// TwinCAT 3 PLC project AbstactDataStructures
// Title: Abstarct Data Structures
// Company: FisoThemes
// Author: Goodwill Mzumala
// Description: Exploring Abstract Data Structures in Structured Text for use in PLCs
// ProgramVersion: 3.1.4022.7
// libraries:
//   Tc2_Standard, * (Beckhoff Automation GmbH)
//   Tc2_System, * (Beckhoff Automation GmbH)
//   Tc2_Utilities, * (Beckhoff Automation GmbH)
//   Tc3_Module, * (Beckhoff Automation GmbH)
//   VisuSymbols,3.5.10.0,System
// project tree:
//   DUTs/Alias/ T_DATA_TYPE.TcDUT (not stored)
//   DUTs/Enum/ E_TYPE_CLASS.TcDUT
//   DUTs/Interface/ I_Stack.TcIO, I_Linked_List.TcIO, I_Queue.TcIO
//   DUTs/Struct/ ST_NODE.TcDUT
//   / GlobalTextList.TcGTLO, PlcTask.TcTTO (not stored)
//   POUs/Dynamic Array/Function Blocks/ FB_Dynamic_Array.TcPOU
//   POUs/Dynamic Array/Programs/ P_Dynamic_Array.TcPOU
//   POUs/Linked List/Function Blocks/ FB_Circular_Linked_List.TcPOU, FB_Doubly_Linked_List.TcPOU, FB_Singly_Linked_List.TcPOU
//   POUs/Linked List/Programs/ P_Doubly_Linked_List.TcPOU, P_Linked_List.TcPOU (not stored), P_Singly_Linked_List.TcPOU
//   POUs/ MAIN.TcPOU
//   POUs/Queue/Function Blocks/ FB_Dynamic_Array_Queue.TcPOU, FB_Linked_List_Queue.TcPOU
//   POUs/Queue/Programs/ P_Dynamic_Array_Queue.TcPOU, P_Linked_List_Queue.TcPOU, P_Queue.TcPOU
//   POUs/Stack/Function Blocks/ FB_Linked_List_Stack.TcPOU, FB_Dynamic_Array_Stack.TcPOU
//   POUs/Stack/Programs/ P_Dynamic_Array_Stack.TcPOU, P_Linked_List_Stack.TcPOU, P_Stack.TcPOU
// real-time tasks:
//   TASK PlcTask: cycle T#10ms, priority 20, ADS port 350

// ---- DUTs/Enum/E_TYPE_CLASS.TcDUT
// List of __SYSTEM.TYPE_CLASS.<type> used for reference
//{attribute 'qualified_only'}
{attribute 'strict'}
TYPE E_TYPE_CLASS :
(
	TYPE_BOOL 			:= DWORD#0,
    TYPE_BIT 			:= DWORD#1,
    TYPE_BYTE 			:= DWORD#2,
    TYPE_WORD 			:= DWORD#3,
    TYPE_DWORD 			:= DWORD#4,
    TYPE_LWORD 			:= DWORD#5,
    TYPE_SINT 			:= DWORD#6,
    TYPE_INT 			:= DWORD#7,
    TYPE_DINT 			:= DWORD#8,
    TYPE_LINT 			:= DWORD#9,
    TYPE_USINT 			:= DWORD#10,
    TYPE_UINT 			:= DWORD#11,
    TYPE_UDINT 			:= DWORD#12,
    TYPE_ULINT 			:= DWORD#13,
    TYPE_REAL 			:= DWORD#14,
    TYPE_LREAL 			:= DWORD#15,
    TYPE_STRING 		:= DWORD#16,
    TYPE_WSTRING 		:= DWORD#17,
    TYPE_TIME 			:= DWORD#18,
    TYPE_DATE 			:= DWORD#19,
    TYPE_DATEANDTIME 	:= DWORD#20,
    TYPE_TIMEOFDAY 		:= DWORD#21,
    TYPE_POINTER 		:= DWORD#22,
    TYPE_REFERENCE 		:= DWORD#23,
    TYPE_SUBRANGE 		:= DWORD#24,
    TYPE_ENUM 			:= DWORD#25,
    TYPE_ARRAY 			:= DWORD#26,
    TYPE_PARAMS 		:= DWORD#27,
    TYPE_USERDEF 		:= DWORD#28,
    TYPE_NONE 			:= DWORD#29,
    TYPE_ANY 			:= DWORD#30,
    TYPE_ANYBIT 		:= DWORD#31,
    TYPE_ANYDATE 		:= DWORD#32,
    TYPE_ANYINT 		:= DWORD#33,
    TYPE_ANYNUM 		:= DWORD#34,
    TYPE_ANYREAL 		:= DWORD#35,
    TYPE_LAZY 			:= DWORD#36,
    TYPE_LTIME 			:= DWORD#37,
    TYPE_BITCONST 		:= DWORD#38
)DWORD;
END_TYPE

// ---- DUTs/Struct/ST_NODE.TcDUT
{attribute 'enable_dynamic_creation'}
TYPE ST_NODE :
STRUCT
	pPrevious 	: POINTER TO ST_NODE := NULL; // Pointer to previos node.
	Data 		: T_DATA_TYPE;
	pNext 		: POINTER TO ST_NODE := NULL; // Pointer to next node.
END_STRUCT
END_TYPE

// ---- DUTs/Interface/I_Stack.TcIO
INTERFACE I_Stack

// Empties/Clears/Deletes all elements on the stack
METHOD Empty
END_METHOD

METHOD FB_exit : BOOL
VAR_INPUT
	bInCopyCode : BOOL; // if TRUE, the exit method is called for exiting an instance that is copied afterwards (online change).
END_VAR
END_METHOD

// Checks of stack is empty.
METHOD Is_Empty : BOOL
VAR_INPUT
END_VAR
END_METHOD

// Gets element at any position of the stack, wuthout removing it.
METHOD Peek : T_DATA_TYPE
VAR_INPUT
	nPosition : DINT;
END_VAR
END_METHOD

// Deletes/pops an element at the front of the stack 
METHOD Pop : T_DATA_TYPE
END_METHOD

// Adds/pushes an element to the front of the stack 
METHOD Push
VAR_INPUT
	Data 	: T_DATA_TYPE;
END_VAR
END_METHOD

// Traverse the stack and display each element as an array
METHOD Show
VAR_IN_OUT
	aList 		: ARRAY[*] OF T_DATA_TYPE; // Array to display data in list.
END_VAR
END_METHOD

// Gets size of the stack
METHOD Size : DINT;
END_METHOD

// Reads/returns the data at the top of the stack without removing it.
METHOD Top : T_DATA_TYPE
VAR_INPUT
END_VAR
END_METHOD

END_INTERFACE

// ---- DUTs/Interface/I_Linked_List.TcIO
INTERFACE I_Linked_List

// Creates/Adds an node to the end of the list
METHOD Create
VAR_INPUT
	Data : T_DATA_TYPE; // Data to add to new node.
END_VAR
END_METHOD

// Empties/Clears/Deletes list
METHOD Empty
END_METHOD

METHOD FB_exit : BOOL
VAR_INPUT
	bInCopyCode : BOOL; // if TRUE, the exit method is called for exiting an instance that is copied afterwards (online change).
END_VAR
END_METHOD

METHOD FB_init : BOOL
VAR_INPUT
	bInitRetains : BOOL; // if TRUE, the retain variables are initialized (warm start / cold start)
	bInCopyCode : BOOL;  // if TRUE, the instance afterwards gets moved into the copy code (online change)
END_VAR
END_METHOD

// Inserts node at a specific position in the list
METHOD Insert
VAR_INPUT
	Data 		: T_DATA_TYPE; 	// Data to add to new node.
	nPosition 	: DINT;		// Position to add new node in list.
END_VAR
END_METHOD

// Checks of list is empty.
METHOD Is_Empty : BOOL
VAR_INPUT
END_VAR
END_METHOD

// Gets element at any position of the list, wuthout removing it.
METHOD Peek : T_DATA_TYPE
VAR_INPUT
	nPosition : DINT;
END_VAR
END_METHOD

// Deletes/pops a node at the front of the list 
METHOD Pop : T_DATA_TYPE
END_METHOD

// Adds/pushes a node at the front of the list 
METHOD Push
VAR_INPUT
		Data 	: T_DATA_TYPE;
END_VAR
END_METHOD

// Deletes node at a specific position in the list
METHOD Remove : T_DATA_TYPE
VAR_INPUT
	nPosition 	: DINT; // Position of node to delete.
END_VAR
END_METHOD

// Reverse list
METHOD Reverse
END_METHOD

// Searches list for the first instance of data and returns it's location and whether it's in the list.
METHOD Search : BOOL
VAR_INPUT
	Data : T_DATA_TYPE; // Data to find in list
END_VAR
VAR_OUTPUT
	nPosition : DINT; // Location of the data  starting from 0. -1 means data is not found in list
END_VAR
END_METHOD

// Traverse the list to display each node
METHOD Show
VAR_IN_OUT
	aList 		: ARRAY[*] OF T_DATA_TYPE; // Array to display data in list.
END_VAR
END_METHOD

// Gets size of the list
METHOD Size : DINT;
END_METHOD

END_INTERFACE

// ---- DUTs/Interface/I_Queue.TcIO
INTERFACE I_Queue

(* Removes element from the front of the queue. *)
METHOD Dequeue : T_DATA_TYPE
VAR_INPUT
END_VAR
END_METHOD

(* Empties/Clears/Deletes all elements on the stack. *)
METHOD Empty
END_METHOD

(* Adds element to the rear of the queue. *)
METHOD Enqueue
VAR_INPUT
	Data 	: T_DATA_TYPE;
END_VAR
END_METHOD

METHOD FB_exit : BOOL
VAR_INPUT
	bInCopyCode : BOOL; // if TRUE, the exit method is called for exiting an instance that is copied afterwards (online change).
END_VAR
END_METHOD

METHOD FB_init : BOOL
VAR_INPUT
	bInitRetains : BOOL; // if TRUE, the retain variables are initialized (warm start / cold start)
	bInCopyCode : BOOL;  // if TRUE, the instance afterwards gets moved into the copy code (online change)
END_VAR
END_METHOD

(* Checks of queue is empty. *)
METHOD Is_Empty : BOOL
VAR_INPUT
END_VAR
END_METHOD

// Gets element at any position of the queue, without removing it.
METHOD Peek : T_DATA_TYPE
VAR_INPUT
	nPosition : DINT;
END_VAR
END_METHOD

(* Traverse the queue and display each element as an array. *)
METHOD Show
VAR_IN_OUT
	aList : ARRAY[*] OF T_DATA_TYPE; // Array to display data in list.
END_VAR
END_METHOD

(* Gets size of the queue. *)
METHOD Size : DINT;
END_METHOD

END_INTERFACE

// ---- POUs/Dynamic Array/Function Blocks/FB_Dynamic_Array.TcPOU
FUNCTION_BLOCK FB_Dynamic_Array
VAR_INPUT
	
END_VAR
VAR_OUTPUT
END_VAR
VAR
	pData 	: POINTER TO T_DATA_TYPE;
	nLength : DINT;
	t_Null	: T_DATA_TYPE;
END_VAR

(* Get element in array from specified poisiton. *)
METHOD Access : T_DATA_TYPE
VAR_INPUT
	nPosition : DINT;  // Position of element in dynamic array, 0 indexed.
END_VAR
IF nPosition < 0 THEN Access := t_Null; RETURN; END_IF
IF THIS^.Is_Empty() THEN FB_Init(FALSE,FALSE,(nPosition+1)*2); END_IF
IF nPosition >= THIS^.Size() THEN THIS^.Insert(t_Null, nPosition); END_IF
Access := THIS^.pData[nPosition];
END_METHOD

(* Deletes array from memory. *)
METHOD Clear
VAR_INPUT
END_VAR
IF NOT(THIS^.Is_Empty()) THEN __DELETE(THIS^.pData); THIS^.Is_Empty(); END_IF
END_METHOD

METHOD FB_exit : BOOL
VAR_INPUT
	bInCopyCode : BOOL; // if TRUE, the exit method is called for exiting an instance that is copied afterwards (online change).
END_VAR
THIS^.Clear();
END_METHOD

METHOD FB_init : BOOL
VAR_INPUT
	bInitRetains 	: BOOL; // if TRUE, the retain variables are initialized (warm start / cold start)
	bInCopyCode 	: BOOL;  // if TRUE, the instance afterwards gets moved into the copy code (online change)
	nLength 		: DINT; 	// Length to initialize array with, default is 10;
END_VAR
THIS^.Clear();
IF nLength > 0 THEN THIS^.pData := __NEW(T_DATA_TYPE, TO_UDINT(nLength)); END_IF
THIS^.nLength := nLength;
END_METHOD

(* Insert element into array at specified position. *)
METHOD Insert
VAR_INPUT
	Data 		: T_DATA_TYPE; 	// Data to insert in dynamic array.
	nPosition 	: DINT; 		// Position to insert data at in the dynamic array, 0 indexed. 
END_VAR
VAR
	pTemp_Data 		: POINTER TO T_DATA_TYPE;
	nTemp_Length 	: DINT;
	i 				: DINT;
END_VAR
IF nPosition < 0 THEN RETURN; END_IF
IF THIS^.Is_Empty() THEN FB_Init(FALSE,FALSE,(nPosition+1)*2); END_IF
IF nPosition < THIS^.Size() THEN 
	THIS^.pData[nPosition] := Data;
ELSE 
	THIS^.Resize((nPosition+1)*2);
	THIS^.pData[nPosition] := Data;
	END_IF
END_METHOD

(* Checks if array is empty. *)
METHOD Is_Empty : BOOL
VAR_INPUT
END_VAR
Is_Empty := THIS^.pData = 0;
IF Is_Empty THEN THIS^.nLength := 0; END_IF
END_METHOD

(* Manually resize dynamic array length. If Array become smaller, elements higher positions will be deleted. *)
METHOD Resize
VAR_INPUT
	nLength 		: DINT; // New length of dynamic array.
END_VAR
VAR_INST
	pTemp_Data 		: POINTER TO T_DATA_TYPE;
	nTemp_Length 	: DINT;
	i 				: DINT;
END_VAR
IF nLength <= 0 THEN THIS^.Clear(); RETURN; END_IF
IF THIS^.Is_Empty() THEN FB_init(FALSE,FALSE,nLength); RETURN; END_IF
IF THIS^.nLength = nLength THEN RETURN; END_IF

pTemp_Data 		:= THIS^.pData; 

nTemp_Length 	:= THIS^.nLength;
THIS^.nLength 	:= nLength;

THIS^.pData := __NEW(T_DATA_TYPE, TO_UDINT(THIS^.nLength));
FOR i := 0 TO TO_DINT(nTemp_Length-1) DO 
	IF i > TO_DINT(THIS^.nLength-1) THEN EXIT; END_IF 
	THIS^.pData[i] := pTemp_Data[i]; 
	END_FOR
__DELETE(pTemp_Data);
END_METHOD

(* Display elements in dynamic array in a static array. *)
METHOD Show
VAR_IN_OUT
	aList : ARRAY[*] OF T_DATA_TYPE; // Static array to display data in dynamic array.
END_VAR
VAR
	i,j : DINT;
END_VAR
FOR i := LOWER_BOUND(aList, 1) TO UPPER_BOUND(aList, 1) DO
	IF (j < TO_DINT(THIS^.Size())) AND NOT(THIS^.Is_Empty()) THEN
		aList[i] := THIS^.pData[j];
		j := j + 1; 
	ELSE 
		aList[i] := t_Null;
	 	END_IF
	END_FOR
END_METHOD

(* Gets the length of dynamic array. *)
METHOD Size : DINT
VAR_INPUT
END_VAR
Is_Empty(); Size := THIS^.nLength;
END_METHOD

END_FUNCTION_BLOCK

// ---- POUs/Dynamic Array/Programs/P_Dynamic_Array.TcPOU
PROGRAM P_Dynamic_Array
VAR
	bIs_Empty, bInsert, bAdd, bAccess, bResize, bClear : BOOL;
	nDyn_Size 	: DINT;
	aArray 		: ARRAY[0..30] OF T_DATA_TYPE;
	t_Access 	: T_DATA_TYPE;  
	fbDyn_Array : FB_Dynamic_Array(10);
	i 			: DINT;
END_VAR

bIs_Empty := fbDyn_Array.Is_Empty();
nDyn_Size := fbDyn_Array.Size();
fbDyn_Array.Show(aArray);

IF bInsert THEN
	fbDyn_Array.Insert(53476,0); 
	FOR i := 1 TO 9 DO fbDyn_Array.Insert(TO_ULINT(i*11),i); END_FOR
	bInsert := 0;
	END_IF
IF bAdd 	THEN fbDyn_Array.Insert(33,10); bAdd 	:= 0; END_IF
IF bAccess 	THEN t_Access := fbDyn_Array.Access(2); bAccess := 0; END_IF
IF bResize 	THEN fbDyn_Array.Resize(5); 			bResize := 0; END_IF
IF bClear 	THEN fbDyn_Array.Clear();				bClear 	:= 0; END_IF

END_PROGRAM

// ---- POUs/Linked List/Function Blocks/FB_Circular_Linked_List.TcPOU
FUNCTION_BLOCK FB_Circular_Linked_List IMPLEMENTS I_Linked_List
VAR_INPUT
END_VAR
VAR_OUTPUT
END_VAR
VAR
END_VAR

{warning 'add method implementation '}
(* Creates/Adds an node to the end of the list*)
METHOD Create
VAR_INPUT
	(* Data to add to new node.*)
	Data	: T_DATA_TYPE;
END_VAR
END_METHOD

{warning 'add method implementation '}
(* Empties/Clears/Deletes list*)
METHOD Empty
	pTemp	: POINTER TO ST_NODE;
END_METHOD

{warning 'add method implementation '}
(* Initializes or create an empty list*)
METHOD Init
END_METHOD

{warning 'add method implementation '}
(* Inserts node at a specific position in the list*)
METHOD Insert
VAR_INPUT
	(* Data to add to new node.*)
	Data	: T_DATA_TYPE;
	(* Position to add new node in list.*)
	nPosition	: UXINT;
END_VAR
END_METHOD

{warning 'add method implementation '}
METHOD Pop
END_METHOD

{warning 'add method implementation '}
METHOD Push
VAR_INPUT
	Data	: T_DATA_TYPE;
END_VAR
END_METHOD

{warning 'add method implementation '}
(* Deletes node at a specific position in the list*)
METHOD Remove
VAR_INPUT
	(* Position of node to delete.*)
	nPosition	: UXINT;
END_VAR
END_METHOD

{warning 'add method implementation '}
(* Searches list for the first instance of data and returns it's location and whether it's in the list.*)
METHOD Search : BOOL
VAR_INPUT
	(* Data to find in list*)
	Data	: T_DATA_TYPE;
END_VAR
VAR_OUTPUT
	(* Location of the data  starting from 1. 0 means data is not found in list*)
	nPosition	: UXINT;
END_VAR
END_METHOD

{warning 'add method implementation '}
METHOD Show
END_METHOD

{warning 'add method implementation '}
(* Gets size of the list*)
METHOD Size : UXINT
END_METHOD

END_FUNCTION_BLOCK

// ---- POUs/Linked List/Function Blocks/FB_Doubly_Linked_List.TcPOU
FUNCTION_BLOCK FB_Doubly_Linked_List IMPLEMENTS I_Linked_List
VAR
	pHead :  POINTER TO ST_NODE;
	pTail :  POINTER TO ST_NODE;
	t_Null: T_DATA_TYPE;
END_VAR

(* Creates/Adds an node to the end of the list. *)
METHOD Create
VAR_INPUT
	(* Data to add to new node.*)
	Data		: T_DATA_TYPE;
END_VAR
VAR
	pTemp 		:  POINTER TO ST_NODE; //  New node will be allocated at this pointer
	pPrevious 	: POINTER TO ST_NODE; // Previous node location will be stored at this pointer temporarily
END_VAR
pTemp := __NEW(ST_NODE);
pTemp^.Data := Data;
IF THIS^.pHead = 0 THEN 
	THIS^.pHead := pTemp; 
	THIS^.pTail := THIS^.pHead; // If the pointer to the pHead is NULL then give it an address. The pTail address of the first node is the pHead.
ELSE
	pPrevious := THIS^.pTail;
	THIS^.pTail^.pNext := pTemp; 
	THIS^.pTail := pTemp;
	THIS^.pTail^.pPrevious := pPrevious; 
	END_IF // Point previous node's pNext to the address of pTemp and set pTail to pTemp.
END_METHOD

(* Empties/Clears/Deletes list*)
METHOD Empty
VAR
	pTemp : POINTER TO ST_NODE;
END_VAR
pTail := 0;
pTemp := pHead;
WHILE pTemp <> 0 DO
	pTemp := pTemp^.pNext; THIS^.Pop();
END_WHILE
END_METHOD

METHOD FB_exit : BOOL
VAR_INPUT
	(* if TRUE, the exit method is called for exiting an instance that is copied afterwards (online change).*)
	bInCopyCode	: BOOL;
END_VAR
This^.Empty();
END_METHOD

METHOD FB_init : BOOL
VAR_INPUT
	(* if TRUE, the retain variables are initialized (warm start / cold start)*)
	bInitRetains	: BOOL;
	(* if TRUE, the instance afterwards gets moved into the copy code (online change)*)
	bInCopyCode	: BOOL;
END_VAR
END_METHOD

(* Inserts node at a specific position in the list*)
METHOD Insert
VAR_INPUT
	(* Data to add to new node.*)
	Data	: T_DATA_TYPE;
	(* Position to add new node in list.*)
	nPosition	: DINT;
END_VAR
END_METHOD

(* Checks of list is empty.*)
METHOD Is_Empty : BOOL
END_METHOD

(* Gets element at any position of the list, wuthout removing it.*)
METHOD Peek : T_DATA_TYPE
VAR_INPUT
	nPosition	: DINT;
END_VAR
END_METHOD

(* Deletes/pops a node at the front of the list *)
METHOD Pop : T_DATA_TYPE
VAR
	pTemp : POINTER TO ST_NODE;
END_VAR
IF THIS^.pHead = 0 THEN RETURN; END_IF 
Pop := pHead^.Data;
pTemp := pHead^.pNext;
__DELETE(pHead);
pHead := pTemp;
END_METHOD

(* Adds/pushes a node at the front of the list *)
METHOD Push
VAR_INPUT
	Data	: T_DATA_TYPE;
END_VAR
END_METHOD

(* Deletes node at a specific position in the list*)
METHOD Remove : T_DATA_TYPE
VAR_INPUT
	(* Position of node to delete.*)
	nPosition	: DINT;
END_VAR
END_METHOD

(* Reverse list*)
METHOD Reverse
END_METHOD

//{warning 'add method implementation '}
(* Searches list for the first instance of data and returns it's location and whether it's in the list.*)
METHOD Search : BOOL
VAR_INPUT
	(* Data to find in list*)
	Data	: T_DATA_TYPE;
END_VAR
VAR_OUTPUT
	(* Location of the data  starting from 1. 0 means data is not found in list*)
	nPosition	: DINT;
END_VAR
END_METHOD

(* Traverse the list to display each node. *)
METHOD Show
VAR_IN_OUT
	aList 		: ARRAY[*] OF T_DATA_TYPE; // Array to display data in list.
END_VAR
VAR
	pCurrent 	: POINTER TO ST_NODE;
	i 			: DINT;
END_VAR
END_METHOD

(* Gets size of the list*)
METHOD Size : DINT
END_METHOD

END_FUNCTION_BLOCK

// ---- POUs/Linked List/Function Blocks/FB_Singly_Linked_List.TcPOU
// Linear/Singly Linked List
FUNCTION_BLOCK FB_Singly_Linked_List IMPLEMENTS I_Linked_List
VAR_INPUT
END_VAR
VAR_OUTPUT
END_VAR
VAR
	pHead :  POINTER TO ST_NODE;
	pTail :  POINTER TO ST_NODE;
	t_Null: T_DATA_TYPE;
END_VAR

// Creates/Adds an node to the end of the list
METHOD Create
VAR_INPUT
	Data : T_DATA_TYPE; // Data to add to new node.
END_VAR
VAR
	pTemp :  POINTER TO ST_NODE;
END_VAR
pTemp := __NEW(ST_NODE); 	// Allocate space in memory for a node.
pTemp^.Data := Data;		// Assign Data to the new node.
IF pHead = 0 THEN pHead := pTemp; pTail := pHead; // If the pointer to the pHead is NULL then give it an address. The pTail address of the first node is the pHead.
ELSE  pTail^.pNext := pTemp; pTail := pTail^.pNext; END_IF // Point previous node's pNext to the address of pTemp and set pTail to pTemp.
END_METHOD

// Empties/Clears/Deletes list
METHOD Empty
VAR
	pTemp : POINTER TO ST_NODE;
END_VAR
pTail := 0;
pTemp := pHead;
WHILE pTemp <> 0 DO
	pTemp := pTemp^.pNext; THIS^.Pop();
END_WHILE
END_METHOD

METHOD FB_exit : BOOL
VAR_INPUT
	bInCopyCode : BOOL; // if TRUE, the exit method is called for exiting an instance that is copied afterwards (online change).
END_VAR
Empty();
END_METHOD

// Initializes or create an empty list
METHOD Init
THIS^.Empty();
pHead := 0;
pTail := 0;
END_METHOD

// Inserts node at a specific position in the list
METHOD Insert
VAR_INPUT
	Data 		: T_DATA_TYPE; 	// Data to add to new node.
	nPosition 	: DINT;		// Position to add new node in list.
END_VAR
VAR
	pPrevious 	: POINTER TO ST_NODE;
	pCurrent 	: POINTER TO ST_NODE;
	pTemp 		: POINTER TO ST_NODE;
	i 			: DINT;
END_VAR
IF nPosition < 0 THEN RETURN; END_IF
IF nPosition = 0 THEN THIS^.Push(Data); RETURN; END_IF
pTemp := __NEW(ST_NODE);
pCurrent := THIS^.pHead;
FOR i := 1 TO nPosition DO // traverse
	pPrevious := pCurrent; 
	pCurrent := pPrevious^.pNext;
	IF pCurrent = 0 THEN EXIT; END_IF
	END_FOR;
pTemp^.Data := Data;
IF pPrevious <> 0 THEN pPrevious^.pNext := pTemp; END_IF
pTemp^.pNext := pCurrent;
END_METHOD

(* Checks of list is empty.*)
METHOD Is_Empty : BOOL
Is_Empty := pHead = 0;
END_METHOD

// Gets element at any position of the list. Returns 0 if element is not found
METHOD Peek : T_DATA_TYPE
VAR_INPUT
	nPosition : DINT;
END_VAR
VAR 
	i 		: DINT;
	pTemp 	: POINTER TO ST_NODE;
END_VAR
IF nPosition >= 0 AND nPosition < THIS^.Size() THEN
	pTemp := pHead;
	FOR i := 0 TO nPosition DO
		Peek := pTemp^.Data;
		pTemp := pTemp^.pNext;
		END_FOR
ELSE
	Peek := 0;
	END_IF
END_METHOD

// Deletes/pops a node at the start of the list 
METHOD Pop : T_DATA_TYPE
VAR
	pTemp : POINTER TO ST_NODE;
END_VAR
IF THIS^.pHead = 0 THEN RETURN; END_IF 
Pop := pHead^.Data;
pTemp := pHead^.pNext;
__DELETE(pHead);
pHead := pTemp;
END_METHOD

// Adds/pushes a node at the start of the list 
METHOD Push
VAR_INPUT
	Data 	: T_DATA_TYPE;
END_VAR
VAR
	pTemp 	:  POINTER TO ST_NODE;
END_VAR
pTemp := __NEW(ST_NODE);
pTemp^.Data := Data;
IF THIS^.pHead = 0 THEN THIS^.pHead := pTemp; THIS^.pTail := THIS^.pHead;
ELSE pTemp^.pNext := THIS^.pHead; THIS^.pHead := pTemp; END_IF
END_METHOD

// Deletes node at a specific position in the list
METHOD Remove : T_DATA_TYPE
VAR_INPUT
	nPosition 	: DINT; // Position of node to delete.
END_VAR
VAR
	pPrevious 	: POINTER TO ST_NODE;
	pCurrent 	: POINTER TO ST_NODE;
	i 			: DINT;
END_VAR
IF nPosition < 0 THEN RETURN; END_IF
pCurrent := pHead;
FOR i := 1 TO nPosition DO
	pPrevious := pCurrent;
	pCurrent := pCurrent^.pNext;
	END_FOR;
Remove := pCurrent^.Data;
pPrevious^.pNext := pCurrent^.pNext;
__DELETE(pCurrent);
END_METHOD

// Reverses list
METHOD Reverse
VAR
	pPrevious 	: POINTER TO ST_NODE;
	pCurrent 	: POINTER TO ST_NODE;
	pNext	 	: POINTER TO ST_NODE;
	i 			: DINT;
END_VAR
pCurrent := pHead;
pNext := pCurrent;
WHILE pCurrent <> 0 DO
	pNext := pNext^.pNext;
	pCurrent^.pNext := pPrevious;
	pPrevious := pCurrent;
	pCurrent := pNext;
END_WHILE
pHead := pPrevious;
END_METHOD

// Searches list for the first instance of data and returns it's location and whether it's in the list.
METHOD Search : BOOL
VAR_INPUT
	Data : T_DATA_TYPE; // Data to find in list
END_VAR
VAR_OUTPUT
	nPosition : DINT; // Location of the data  starting from 1. 0 means data is not found in list
END_VAR
VAR
	pTemp 	: POINTER TO ST_NODE;
	i 		: DINT;
END_VAR
pTemp := pHead;
WHILE pTemp <> 0 DO
	
	Search := pTemp^.Data = Data;
	IF Search THEN nPosition := i; EXIT; ELSE nPosition := 0; END_IF
	i := i + 1;
	pTemp := pTemp^.pNext;
END_WHILE
END_METHOD

// Traverse the list to display each node
METHOD Show
VAR_IN_OUT
	aList 		: ARRAY[*] OF T_DATA_TYPE; // Array to display data in list.
END_VAR
VAR
	pCurrent 	: POINTER TO ST_NODE;
	i 			: DINT;
END_VAR
pCurrent := THIS^.pHead;
FOR i := LOWER_BOUND(aList, 1) TO UPPER_BOUND(aList, 1) DO
	IF pCurrent <> 0 THEN 
		aList[i] := pCurrent^.Data; 
		pCurrent := pCurrent^.pNext;
	ELSE
		aList[i] := t_Null;
		END_IF
	END_FOR
END_METHOD

// Gets size of the list
METHOD Size : DINT;
VAR
	pTemp 	: POINTER TO ST_NODE;
	i 		: dINT;
END_VAR
pTemp := pHead;
WHILE pTemp <> 0 DO
	pTemp := pTemp^.pNext; i := i + 1;;
END_WHILE
Size := i;
END_METHOD

END_FUNCTION_BLOCK

// ---- POUs/Linked List/Programs/P_Doubly_Linked_List.TcPOU
PROGRAM P_Doubly_Linked_List
VAR
	nState 			: BYTE;
	fbLinked_List 	: FB_Doubly_Linked_List;
	Peek 			: T_DATA_TYPE;
	
	bFound 			: BOOL;		// Is data in the created list?
	nPosition 		: DINT;	// At what position is the data on the list? 0 means no data found. Head mode is 1.
	
	nSize 			: DINT; 	// Dispays size of list after it's created
	nDelete_Size 	: DINT; 	// Displays size of list after deleting an element.
	nInsert_Size 	: DINT; 	// Displays size of list after inserting an element.
	
	aArray 			: ARRAY[1..6] OF T_DATA_TYPE; // Displays created list.
	aDelete_Array 	: ARRAY[1..6] OF T_DATA_TYPE; // Displays list after deleting element at a position.
	aInsert_Array	: ARRAY[1..6] OF T_DATA_TYPE; // Displays list after inserting element at a position.
END_VAR

CASE nState OF 
	0: // Create list, display list, get list size and find an item in the list.
		fbLinked_List.Create(1);
		fbLinked_List.Create(2);
		fbLinked_List.Create(3);
		fbLinked_List.Create(4);
		fbLinked_List.Create(5);
		fbLinked_List.Show(aArray);
		Peek := fbLinked_List.Peek(1);
		nSize := fbLinked_List.Size();
		bFound := fbLinked_List.Search(Data := 5, nPosition => nPosition);

		nState := nState + 1;			
	
	1: // Remove an elements from the list, display list and get the list size
		fbLinked_list.Remove(3);
		fbLinked_List.Pop();
		fbLinked_List.Show(aDelete_Array);
		nDelete_Size := fbLinked_List.Size();
	
		nState := nState + 1;
	
	2: // Insert elements into list, display it and the list size
		fbLinked_List.Push(11);
		fbLinked_List.Insert(14,3);
		fbLinked_List.Show(aInsert_Array);
		nInsert_Size := fbLinked_List.Size();
		
		nState := nState + 1;
		
	3: // Clear list, then finish.
		fbLinked_List.Empty();
		
		nState := nState + 1;
END_CASE

END_PROGRAM

// ---- POUs/Linked List/Programs/P_Singly_Linked_List.TcPOU
PROGRAM P_Singly_Linked_List
VAR
	nState 			: BYTE;
	fbLinked_List 	: FB_Singly_Linked_List;
	Peek 			: T_DATA_TYPE;
	
	bFound 			: BOOL;		// Is data in the created list?
	nPosition 		: DINT;	// At what position is the data on the list? 0 means no data found. Head mode is 1.
	
	nCreate_Size 	: DINT; 	// Dispays size of list after it's created
	nDelete_Size 	: DINT; 	// Displays size of list after deleting an element.
	nInsert_Size 	: DINT; 	// Displays size of list after inserting an element.
	nClear_Size 	: DINT; 	// Displays size of list after clearing all elements.
	
	aCreate_Array 	: ARRAY[1..6] OF T_DATA_TYPE; // Displays created list.
	aDelete_Array 	: ARRAY[1..6] OF T_DATA_TYPE; // Displays list after deleting element at a position.
	aInsert_Array	: ARRAY[1..6] OF T_DATA_TYPE; // Displays list after inserting element at a position.
	aClear_Array	: ARRAY[1..6] OF T_DATA_TYPE; // Displays list after clearing all elements.
	
	
END_VAR

CASE nState OF 
	0: // Create list, display list, get list size and find an item in the list.
		fbLinked_List.Create(1);
		fbLinked_List.Create(2);
		fbLinked_List.Create(3);
		fbLinked_List.Create(4);
		fbLinked_List.Create(5);
		fbLinked_List.Show(aCreate_Array);
		Peek := fbLinked_List.Peek(1);
		nCreate_Size := fbLinked_List.Size();
		bFound := fbLinked_List.Search(Data := 5, nPosition => nPosition);

		nState := nState + 1;			
	
	1: // Remove an elements from the list, display list and get the list size
		fbLinked_list.Remove(3);
		fbLinked_List.Pop();
		fbLinked_List.Show(aDelete_Array);
		nDelete_Size := fbLinked_List.Size();
	
		nState := nState + 1;
	
	2: // Insert elements into list, display it and the list size
		fbLinked_List.Push(11);
		fbLinked_List.Insert(14,3);
		fbLinked_List.Show(aInsert_Array);
		nInsert_Size := fbLinked_List.Size();
		
		nState := nState + 1;
		
	3: // Clear list, then finish.
		fbLinked_List.Empty();
		fbLinked_List.Show(aClear_Array);
		nClear_Size := fbLinked_List.Size();
		
		nState := nState + 1;
END_CASE

END_PROGRAM

// ---- POUs/MAIN.TcPOU
PROGRAM MAIN
VAR
END_VAR

P_Dynamic_Array();
P_Linked_List();
P_Queue();
P_Stack();

END_PROGRAM

// ---- POUs/Queue/Programs/P_Queue.TcPOU
PROGRAM P_Queue
VAR
END_VAR

P_Dynamic_Array_Queue();
P_Linked_List_Queue();

END_PROGRAM

// ---- POUs/Queue/Programs/P_Dynamic_Array_Queue.TcPOU
PROGRAM P_Dynamic_Array_Queue
VAR
	nState 	: BYTE;
	fbQueue : FB_Dynamic_Array_Queue;
	
	bInit_Is_Empty 		: BOOL;
	nInit_Size 			: DINT;
	Init_Peek 			: T_DATA_TYPE;
	aInit_Show 			: ARRAY[1..6] OF T_DATA_TYPE;
	
	bEnqueue_Is_Empty 	: BOOL;
	nEnqueue_Size 		: DINT;
	Enqueue_Peek 		: T_DATA_TYPE;
	aEnqueue_Show 		: ARRAY[1..6] OF T_DATA_TYPE;
	
	bDequeue_Is_Empty 	: BOOL;
	nDequeue_Size 		: DINT;
	Dequeue_Peek 		: T_DATA_TYPE;
	aDequeue_Show 		: ARRAY[1..6] OF T_DATA_TYPE;
	
	bEmpty_Is_Empty 	: BOOL;
	nEmpty_Size 		: DINT;
	Empty_Peek 			: T_DATA_TYPE;
	aEmpty_Show 		: ARRAY[1..6] OF T_DATA_TYPE;
END_VAR

CASE nState OF
	0: // Init
		bInit_Is_Empty := fbQueue.Is_Empty();
		nInit_Size :=  fbQueue.Size();
		Init_Peek := fbQueue.Peek(0);
		fbQueue.Show(aInit_Show);
		
		nState := nState + 1;
		
	1: // Enqueue elements
		fbQueue.Enqueue(1);
		fbQueue.Enqueue(2);
		fbQueue.Enqueue(3);
		fbQueue.Enqueue(4);
		fbQueue.Enqueue(5);
		bEnqueue_Is_Empty := fbQueue.Is_Empty();
		nEnqueue_Size := fbQueue.Size();
		Enqueue_Peek := fbQueue.Peek(0);
		fbQueue.Show(aEnqueue_Show);
		
		nState := nState + 1;
	
	2: // Dequeue elements
		fbQueue.Dequeue();
		fbQueue.Dequeue(); 
		bDequeue_Is_Empty := fbQueue.Is_Empty();
		nDequeue_Size := fbQueue.Size();
		Dequeue_Peek := fbQueue.Peek(0);
		fbQueue.Show(aDequeue_Show);
		
		nState := nState + 1;
	
	3: // Empty Queue
		fbQueue.Empty();
		bEmpty_Is_Empty := fbQueue.Is_Empty();
		nEmpty_Size := fbQueue.Size();
		Empty_Peek := fbQueue.Peek(0);
		fbQueue.Show(aEmpty_Show);
		
		nState := nState + 1;
	
END_CASE

END_PROGRAM

// ---- POUs/Queue/Function Blocks/FB_Dynamic_Array_Queue.TcPOU
FUNCTION_BLOCK FB_Dynamic_Array_Queue IMPLEMENTS I_Queue
VAR
	fbDynamic_Array : FB_Dynamic_Array(10);
	nSize 			: DINT;
END_VAR

(* Removes element from the front of the queue. *)
METHOD Dequeue : T_DATA_TYPE
VAR 
	i : DINT;
END_VAR
Dequeue := THIS^.fbDynamic_Array.Access(0);
IF THIS^.Is_Empty() THEN RETURN; END_IF
nSize := THIS^.Size() - 1;
FOR i := 1 TO THIS^.nSize DO
	THIS^.fbDynamic_Array.Insert(THIS^.fbDynamic_Array.Access(i),i-1);
	END_FOR
END_METHOD

(* Empties/Clears/Deletes all elements on the stack. *)
METHOD Empty
THIS^.fbDynamic_Array.Clear(); 
THIS^.nSize := THIS^.fbDynamic_Array.Size();
END_METHOD

(* Adds element to the rear of the queue. *)
METHOD Enqueue
VAR_INPUT
	Data	: T_DATA_TYPE;
END_VAR
nSize := THIS^.Size() + 1;
THIS^.fbDynamic_Array.Insert(Data, THIS^.Size()-1);
END_METHOD

METHOD FB_exit : BOOL
VAR_INPUT
	(* if TRUE, the exit method is called for exiting an instance that is copied afterwards (online change).*)
	bInCopyCode	: BOOL;
END_VAR
THIS^.Empty();
END_METHOD

METHOD FB_init : BOOL
VAR_INPUT
	(* if TRUE, the retain variables are initialized (warm start / cold start)*)
	bInitRetains	: BOOL;
	(* if TRUE, the instance afterwards gets moved into the copy code (online change)*)
	bInCopyCode	: BOOL;
END_VAR
END_METHOD

(* Checks of queue is empty. *)
METHOD Is_Empty : BOOL
Is_Empty := nSize = 0;
IF Is_Empty THEN THIS^.Empty(); END_IF
END_METHOD

(* Gets element at any position of the queue, without removing it.*)
METHOD Peek : T_DATA_TYPE
VAR_INPUT
	nPosition	: DINT;
END_VAR
IF (nPosition > THIS^.nSize - 1) THEN nPosition := -1; END_IF
Peek := THIS^.fbDynamic_Array.Access(nPosition);
END_METHOD

(* Traverse the queue and display each element as an array. *)
METHOD Show
VAR_IN_OUT
	aList : ARRAY[*] OF T_DATA_TYPE; // Array to display data in list.
END_VAR
VAR
	i,j : DINT;
END_VAR
FOR i := LOWER_BOUND(aList, 1) TO UPPER_BOUND(aList, 1) DO
	IF j < TO_DINT(THIS^.Size()) AND NOT(THIS^.Is_Empty())THEN 
		aList[i] := THIS^.fbDynamic_Array.Access(j);
		j := j + 1;
	ELSE 
		aList[i] := THIS^.fbDynamic_Array.Access(-1);
		END_IF
	END_FOR
END_METHOD

(* Gets size of the queue. *)
METHOD Size : DINT
IF NOT(THIS^.Is_Empty())THEN Size := THIS^.nSize; END_IF
END_METHOD

END_FUNCTION_BLOCK

// ---- POUs/Queue/Programs/P_Linked_List_Queue.TcPOU
PROGRAM P_Linked_List_Queue
VAR
	nState 	: BYTE;
	fbQueue : FB_Linked_List_Queue;
	
	bInit_Is_Empty 		: BOOL;
	nInit_Size 			: DINT;
	Init_Peek 			: T_DATA_TYPE;
	aInit_Show 			: ARRAY[1..6] OF T_DATA_TYPE;
	
	bEnqueue_Is_Empty 	: BOOL;
	nEnqueue_Size 		: DINT;
	Enqueue_Peek 		: T_DATA_TYPE;
	aEnqueue_Show 		: ARRAY[1..6] OF T_DATA_TYPE;
	
	bDequeue_Is_Empty 	: BOOL;
	nDequeue_Size 		: DINT;
	Dequeue_Peek 		: T_DATA_TYPE;
	aDequeue_Show 		: ARRAY[1..6] OF T_DATA_TYPE;
	
	bEmpty_Is_Empty 	: BOOL;
	nEmpty_Size 		: DINT;
	Empty_Peek 			: T_DATA_TYPE;
	aEmpty_Show 		: ARRAY[1..6] OF T_DATA_TYPE;
END_VAR

CASE nState OF
	0: // Init
		bInit_Is_Empty := fbQueue.Is_Empty();
		nInit_Size :=  fbQueue.Size();
		Init_Peek := fbQueue.Peek(0);
		fbQueue.Show(aInit_Show);
		
		nState := nState + 1;
		
	1: // Enqueue elements
		fbQueue.Enqueue(1);
		fbQueue.Enqueue(2);
		fbQueue.Enqueue(3);
		fbQueue.Enqueue(4);
		fbQueue.Enqueue(5);
		bEnqueue_Is_Empty := fbQueue.Is_Empty();
		nEnqueue_Size := fbQueue.Size();
		Enqueue_Peek := fbQueue.Peek(0);
		fbQueue.Show(aEnqueue_Show);
		
		nState := nState + 1;
	
	2: // Dequeue elements
		fbQueue.Dequeue();
		fbQueue.Dequeue(); 
		bDequeue_Is_Empty := fbQueue.Is_Empty();
		nDequeue_Size := fbQueue.Size();
		Dequeue_Peek := fbQueue.Peek(0);
		fbQueue.Show(aDequeue_Show);
		
		nState := nState + 1;
	
	3: // Empty Queue
		fbQueue.Empty();
		bEmpty_Is_Empty := fbQueue.Is_Empty();
		nEmpty_Size := fbQueue.Size();
		Empty_Peek := fbQueue.Peek(0);
		fbQueue.Show(aEmpty_Show);
		
		nState := nState + 1;
	
END_CASE

END_PROGRAM

// ---- POUs/Queue/Function Blocks/FB_Linked_List_Queue.TcPOU
FUNCTION_BLOCK FB_Linked_List_Queue IMPLEMENTS I_Queue
VAR
	fbLinked_List : FB_Singly_Linked_List;
END_VAR

(* Removes element from the front of the queue. *)
METHOD Dequeue : T_DATA_TYPE
Dequeue := THIS^.fbLinked_List.Pop();
END_METHOD

(* Empties/Clears/Deletes all elements on the stack. *)
METHOD Empty
THIS^.fbLinked_List.Empty();
END_METHOD

(* Adds element to the rear of the queue. *)
METHOD Enqueue
VAR_INPUT
	Data	: T_DATA_TYPE;
END_VAR
THIS^.fbLinked_List.Create(Data);
END_METHOD

METHOD FB_exit : BOOL
VAR_INPUT
	(* if TRUE, the exit method is called for exiting an instance that is copied afterwards (online change).*)
	bInCopyCode	: BOOL;
END_VAR
THIS^.Empty();
END_METHOD

METHOD FB_init : BOOL
VAR_INPUT
	(* if TRUE, the retain variables are initialized (warm start / cold start)*)
	bInitRetains	: BOOL;
	(* if TRUE, the instance afterwards gets moved into the copy code (online change)*)
	bInCopyCode	: BOOL;
END_VAR
END_METHOD

(* Checks of queue is empty. *)
METHOD Is_Empty : BOOL
Is_Empty := THIS^.fbLinked_List.Is_Empty();
END_METHOD

(* Gets element at any position of the queue, without removing it.*)
METHOD Peek : T_DATA_TYPE
VAR_INPUT
	nPosition	: DINT;
END_VAR
Peek := THIS^.fbLinked_List.Peek(nPosition);
END_METHOD

(* Traverse the queue and display each element as an array. *)
METHOD Show
VAR_IN_OUT
	aList :  ARRAY[*] OF T_DATA_TYPE; // Array to display data in list.
END_VAR
THIS^.fbLinked_List.Show(aList);
END_METHOD

(* Gets size of the queue. *)
METHOD Size : DINT
Size := THIS^.fbLinked_List.Size();
END_METHOD

END_FUNCTION_BLOCK

// ---- POUs/Stack/Programs/P_Stack.TcPOU
PROGRAM P_Stack
VAR
END_VAR

P_Dynamic_Array_Stack();
P_Linked_List_Stack();

END_PROGRAM

// ---- POUs/Stack/Programs/P_Dynamic_Array_Stack.TcPOU
PROGRAM P_Dynamic_Array_Stack
VAR
	nState 	: BYTE;
	fbStack : FB_Dynamic_Array_Stack;
	
	
	// Init
	bInit_Is_Empty 	: BOOL;
	nInit_Size 		: DINT;
	Init_Top 		: T_DATA_TYPE;
	aInit_Stack 	: ARRAY[1..6] OF T_DATA_TYPE;
	
	// Pust element to stack
	bPush_Is_Empty 	: BOOL;
	nPush_Size 		: DINT;
	Push_Top 		: T_DATA_TYPE;
	Push_Peek		: T_DATA_TYPE;
	aPush_Stack 	: ARRAY[1..6] OF T_DATA_TYPE; 
	
	// Pop element from stack
	bPop_Is_Empty 	: BOOL;
	nPop_Size 		: DINT;
	Pop_Top 		: T_DATA_TYPE;
	aPop_Stack 		: ARRAY[1..6] OF T_DATA_TYPE; 
	
	// Empty Stack
	bEmpty_Is_Empty : BOOL;
	nEmpty_Size 	: DINT;
	Empty_Top 		: T_DATA_TYPE;
	aEmpty_Stack 	: ARRAY[1..6] OF T_DATA_TYPE; 
END_VAR

CASE nState OF
	0: // Init
		bInit_Is_Empty := fbStack.Is_Empty();
		nInit_Size :=  fbStack.Size();
		Init_Top := fbStack.Top();
		fbStack.Show(aInit_Stack);
		
		nState := nState + 1;
		
	1: // Push Element to tack
		fbStack.Push(1);
		fbStack.Push(2);
		fbStack.Push(3);
		fbStack.Push(4);
		fbStack.Push(5);
		bPush_Is_Empty := fbStack.Is_Empty();
		nPush_Size := fbStack.Size();
		Push_Top := fbStack.Top();
		Push_Peek := fbStack.Peek(2);
		fbStack.Show(aPush_Stack);
		
		nState := nState + 1;
	
	2: // Pop elements from stack
		fbStack.Pop();
		fbStack.Pop();
		bPop_Is_Empty := fbStack.Is_Empty();
		nPop_Size := fbStack.Size();
		Pop_Top := fbStack.Top();
		fbStack.Show(aPop_Stack);
		
		nState := nState + 1;
		
	3: // Empty stack
		fbStack.Empty();
		bEmpty_Is_Empty := fbStack.Is_Empty();
		nEmpty_Size := fbStack.Size();
		Empty_Top := fbStack.Top();
		fbStack.Show(aEmpty_Stack);
		
		nState := nState + 1;
END_CASE

END_PROGRAM

// ---- POUs/Stack/Function Blocks/FB_Dynamic_Array_Stack.TcPOU
FUNCTION_BLOCK FB_Dynamic_Array_Stack IMPLEMENTS I_Stack
VAR_INPUT
END_VAR
VAR_OUTPUT
END_VAR
VAR
	fbDynamic_Array : FB_Dynamic_Array(10); 
	nTop_Index 		: DINT; 
	nSize 			: DINT;
	t_Null 			: T_DATA_TYPE;
END_VAR

(* Empties/Clears/Deletes all elements on the stack*)
METHOD Empty
THIS^.fbDynamic_Array.Clear(); 
THIS^.nSize := THIS^.fbDynamic_Array.Size();
END_METHOD

METHOD FB_exit : BOOL
VAR_INPUT
	(* if TRUE, the exit method is called for exiting an instance that is copied afterwards (online change).*)
	bInCopyCode	: BOOL;
END_VAR
THIS^.Empty();
END_METHOD

METHOD FB_init : BOOL
VAR_INPUT
	bInitRetains : BOOL; // if TRUE, the retain variables are initialized (warm start / cold start)
	bInCopyCode : BOOL;  // if TRUE, the instance afterwards gets moved into the copy code (online change)
END_VAR
END_METHOD

(* Checks of stack is empty.*)
METHOD Is_Empty : BOOL
Is_Empty := nSize = 0;
IF Is_Empty THEN THIS^.Empty(); END_IF
END_METHOD

(* Gets element at any position of the stack, without removing it.*)
METHOD Peek : T_DATA_TYPE
VAR_INPUT
	nPosition	: DINT;
END_VAR
IF (nPosition > THIS^.nSize - 1) THEN nPosition := -1; END_IF
Peek := THIS^.fbDynamic_Array.Access(nPosition);
END_METHOD

(* Deletes/pops an element at the front of the stack *)
METHOD Pop : T_DATA_TYPE
Pop := THIS^.fbDynamic_Array.Access(THIS^.Size() - 1);
IF NOT(THIS^.Is_Empty()) THEN nSize := THIS^.Size() - 1; END_IF
END_METHOD

(* Adds/pushes an element to the front of the stack *)
METHOD Push
VAR_INPUT
	Data	: T_DATA_TYPE;
END_VAR
nSize := THIS^.Size() + 1;
THIS^.fbDynamic_Array.Insert(Data, THIS^.Size()-1);
END_METHOD

(* Traverse the stack and display each element as an array. *)
METHOD Show
VAR_IN_OUT
	aList : ARRAY[*] OF T_DATA_TYPE; // Array to display data in list.
END_VAR
VAR
	i,j : DINT;
END_VAR
FOR i := LOWER_BOUND(aList, 1) TO UPPER_BOUND(aList, 1) DO
	IF j < TO_DINT(THIS^.Size()) AND NOT(THIS^.Is_Empty())THEN 
		aList[i] := THIS^.fbDynamic_Array.Access((THIS^.Size()-1) - j);
		j := j + 1;
	ELSE 
		aList[i] := THIS^.fbDynamic_Array.Access(-1); 
		END_IF
	END_FOR
END_METHOD

(* Gets size of the stack*)
METHOD Size : DINT
IF NOT(THIS^.Is_Empty())THEN Size := THIS^.nSize; END_IF
END_METHOD

(* Reads/returns the data at the top of the stack without removing it. *)
METHOD Top : T_DATA_TYPE
IF NOT(THIS^.Is_Empty()) THEN Top := THIS^.fbDynamic_Array.Access(THIS^.nSize-1); END_IF
END_METHOD

END_FUNCTION_BLOCK

// ---- POUs/Stack/Programs/P_Linked_List_Stack.TcPOU
PROGRAM P_Linked_List_Stack
VAR
	nState 	: BYTE;
	fbStack : FB_Linked_List_Stack;
	
	
	// Init
	bInit_Is_Empty 	: BOOL;
	nInit_Size 		: DINT;
	Init_Top 		: T_DATA_TYPE;
	aInit_Stack 	: ARRAY[1..6] OF T_DATA_TYPE;
	
	// Pust element to stack
	bPush_Is_Empty 	: BOOL;
	nPush_Size 		: DINT;
	Push_Top 		: T_DATA_TYPE;
	Push_Peek		: T_DATA_TYPE;
	aPush_Stack 	: ARRAY[1..6] OF T_DATA_TYPE; 
	
	// Pop element from stack
	bPop_Is_Empty 	: BOOL;
	nPop_Size 		: DINT;
	Pop_Top 		: T_DATA_TYPE;
	aPop_Stack 		: ARRAY[1..6] OF T_DATA_TYPE; 
	
	// Empty Stack
	bEmpty_Is_Empty : BOOL;
	nEmpty_Size 	: DINT;
	Empty_Top 		: T_DATA_TYPE;
	aEmpty_Stack 	: ARRAY[1..6] OF T_DATA_TYPE; 
END_VAR

CASE nState OF
	0: // Init
		bInit_Is_Empty := fbStack.Is_Empty();
		nInit_Size :=  fbStack.Size();
		Init_Top := fbStack.Top();
		fbStack.Show(aInit_Stack);
		
		nState := nState + 1;
		
	1: // Push Element to tack
		fbStack.Push(1);
		fbStack.Push(2);
		fbStack.Push(3);
		fbStack.Push(4);
		fbStack.Push(5);
		bPush_Is_Empty := fbStack.Is_Empty();
		nPush_Size := fbStack.Size();
		Push_Top := fbStack.Top();
		Push_Peek := fbStack.Peek(2);
		fbStack.Show(aPush_Stack);
		
		nState := nState + 1;
	
	2: // Pop elements from stack
		fbStack.Pop();
		fbStack.Pop();
		bPop_Is_Empty := fbStack.Is_Empty();
		nPop_Size := fbStack.Size();
		Pop_Top := fbStack.Top();
		fbStack.Show(aPop_Stack);
		
		nState := nState + 1;
		
	3: // Empty stack
		fbStack.Empty();
		bEmpty_Is_Empty := fbStack.Is_Empty();
		nEmpty_Size := fbStack.Size();
		Empty_Top := fbStack.Top();
		fbStack.Show(aEmpty_Stack);
		
		nState := nState + 1;
END_CASE

END_PROGRAM

// ---- POUs/Stack/Function Blocks/FB_Linked_List_Stack.TcPOU
FUNCTION_BLOCK FB_Linked_List_Stack IMPLEMENTS I_Stack
VAR
	fbLinked_List : FB_Singly_Linked_List;
	t_Null: T_DATA_TYPE;
END_VAR

(* Empties/Clears/Deletes all elements on the stack*)
METHOD Empty
THIS^.fbLinked_List.Empty();
END_METHOD

METHOD FB_exit : BOOL
VAR_INPUT
	(* if TRUE, the exit method is called for exiting an instance that is copied afterwards (online change).*)
	bInCopyCode	: BOOL;
END_VAR
THIS^.Empty();
END_METHOD

(* Checks of stack is empty.*)
METHOD Is_Empty : BOOL
Is_Empty := THIS^.fbLinked_List.Is_Empty();
END_METHOD

(* Gets element at any position of the stack, wuthout removing it.*)
METHOD Peek : T_DATA_TYPE
VAR_INPUT
	nPosition	: DINT;
END_VAR
Peek := THIS^.fbLinked_List.Peek(nPosition);
END_METHOD

(* Deletes/pops an element at the front of the stack *)
METHOD Pop : T_DATA_TYPE
Pop := THIS^.fbLinked_List.Pop();
END_METHOD

(* Adds/pushes an element to the front of the stack *)
METHOD Push
VAR_INPUT
	Data	: T_DATA_TYPE;
END_VAR
THIS^.fbLinked_List.Push(Data);
END_METHOD

(* Traverse the stack and display each element as an array*)
METHOD Show
VAR_IN_OUT
	aList : ARRAY[*] OF T_DATA_TYPE; // Array to display data in list.
END_VAR
THIS^.fbLinked_List.Show(aList);
END_METHOD

(* Gets size of the list*)
METHOD Size : DINT
Size := THIS^.fbLinked_List.Size();
END_METHOD

(* Reads/returns the data at the top of the stack without removing it. *)
METHOD Top : T_DATA_TYPE
IF THIS^.Is_Empty() THEN Top :=Top := THIS^.fbLinked_List.Peek(-1); ELSE Top := THIS^.fbLinked_List.Peek(0); END_IF
END_METHOD

END_FUNCTION_BLOCK

// ---- GlobalTextList.TcGTLO
TEXTLIST GlobalTextList
  613 = 'cars'
END_TEXTLIST
